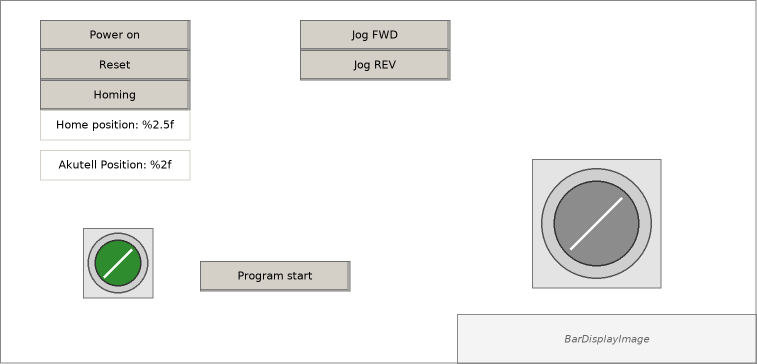
VISUALIZATION Visualization  // 757x364
    Potentiometer360 (524,159 145x129), variable: GVL_Motion.lrSA_PowerOverride, style: Potentiometer-Potentiometer360-Gray, scale format: %.1f, scale 0..100
        p2431819421: Outside
    BarDisplayImage (457,314 300x50), value: GVL_Motion.lrSA_PowerOverride, style: BarDisplayImage-Gray, scale format: %.1f, scale 0..100
    Button (40,20 150x30), "Power on"
        toggle GVL_Motion.bSA_PowerEnCmd
    Button (300,20 150x30), "Jog FWD"
        tap GVL_Motion.bSA_JogFwd
    Button (300,50 150x30), "Jog REV"
        tap GVL_Motion.bSA_JogRev
    Textfield (40,150 150x30), "Akutell Position: %2f", text variable: GVL_Motion.Y_Axis.NcToPlc.ActPos
    Button (40,50 150x30), "Reset"
        tap GVL_Motion.bSA_ResetExe
    Button (40,80 150x30), "Homing"
        tap GVL_Motion.bSA_HomeExe
    Textfield (40,110 150x30), "Home position: %2.5f", text variable: GVL_Motion.lrSA_HomePosition
    RotarySwitch (83,228 70x70), variable: GVL.bAutomaticMode, behaviour: TOGGLE, style: Switch-RotarySwitch-Green
    Button (200,261 150x30), "Program start"
        tap GVL.bKapsekvens
END_VISUALIZATION

(* stored: Version 1.1.0.1, ProductVersion 3.1.4024.10
   Visu Visualization: Id {6ddb2026-f1cf-4d9e-8ec3-b4844b2880eb} *)
